FUNCTION_BLOCK fb_operationElecylinder
VAR_INPUT
END_VAR
VAR_OUTPUT
END_VAR
VAR
	SFCInit: bool;
	TranPosDone: BOOL;
	TranNegDone: BOOL;
	SamplePosDone: BOOL;
	SampleNegDone: BOOL;
	TrayChangePosDone: BOOL;
	TrayChangeNegDone: BOOL;
	flgInitDone: BOOL;
	trn_RotaryNegDone: BOOL;
	trn_RotaryPosDone: BOOL;
	trn_flgInitDone: BOOL;
	var_process: INT;
END_VAR

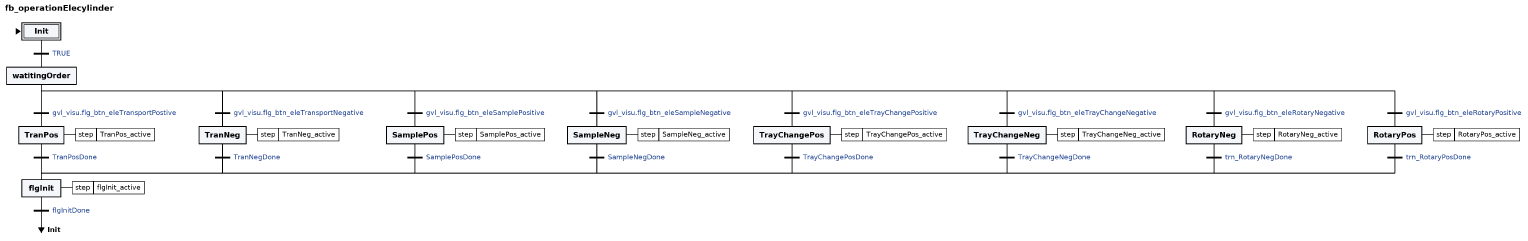
INITIAL_STEP Init:
END_STEP
TRANSITION FROM Init TO watitingOrder
    := TRUE;
END_TRANSITION
STEP watitingOrder:
END_STEP
TRANSITION FROM watitingOrder TO TranPos
    := gvl_visu.flg_btn_eleTransportPostive;
END_TRANSITION
STEP TranPos:
    TranPos_active(N);  // step action
END_STEP
TRANSITION FROM TranPos TO flgInit
    := TranPosDone;
END_TRANSITION
TRANSITION FROM watitingOrder TO TranNeg
    := gvl_visu.flg_btn_eleTransportNegative;
END_TRANSITION
STEP TranNeg:
    TranNeg_active(N);  // step action
END_STEP
TRANSITION FROM TranNeg TO flgInit
    := TranNegDone;
END_TRANSITION
TRANSITION FROM watitingOrder TO SamplePos
    := gvl_visu.flg_btn_eleSamplePositive;
END_TRANSITION
STEP SamplePos:
    SamplePos_active(N);  // step action
END_STEP
TRANSITION FROM SamplePos TO flgInit
    := SamplePosDone;
END_TRANSITION
TRANSITION FROM watitingOrder TO SampleNeg
    := gvl_visu.flg_btn_eleSampleNegative;
END_TRANSITION
STEP SampleNeg:
    SampleNeg_active(N);  // step action
END_STEP
TRANSITION FROM SampleNeg TO flgInit
    := SampleNegDone;
END_TRANSITION
TRANSITION FROM watitingOrder TO TrayChangePos
    := gvl_visu.flg_btn_eleTrayChangePositive;
END_TRANSITION
STEP TrayChangePos:
    TrayChangePos_active(N);  // step action
END_STEP
TRANSITION FROM TrayChangePos TO flgInit
    := TrayChangePosDone;
END_TRANSITION
TRANSITION FROM watitingOrder TO TrayChangeNeg
    := gvl_visu.flg_btn_eleTrayChangeNegative;
END_TRANSITION
STEP TrayChangeNeg:
    TrayChangeNeg_active(N);  // step action
END_STEP
TRANSITION FROM TrayChangeNeg TO flgInit
    := TrayChangeNegDone;
END_TRANSITION
TRANSITION FROM watitingOrder TO RotaryNeg
    := gvl_visu.flg_btn_eleRotaryNegative;
END_TRANSITION
STEP RotaryNeg:
    RotaryNeg_active(N);  // step action
END_STEP
TRANSITION FROM RotaryNeg TO flgInit
    := trn_RotaryNegDone;
END_TRANSITION
TRANSITION FROM watitingOrder TO RotaryPos
    := gvl_visu.flg_btn_eleRotaryPositive;
END_TRANSITION
STEP RotaryPos:
    RotaryPos_active(N);  // step action
END_STEP
TRANSITION FROM RotaryPos TO flgInit
    := trn_RotaryPosDone;
END_TRANSITION
STEP flgInit:
    flgInit_active(N);  // step action
END_STEP
TRANSITION FROM flgInit TO Init
    := flgInitDone;
END_TRANSITION

ACTION flgInit_active:
IF flgInit._x AND flgInit.x = FALSE THEN
	flgInitDone:= FALSE;
	gvl_visu.flg_btn_eleTransportPostive := FALSE;
	gvl_visu.flg_btn_eleTransportNegative := FALSE;
	gvl_visu.flg_btn_eleSamplePositive := FALSE;
	gvl_visu.flg_btn_eleSampleNegative := FALSE;
	gvl_visu.flg_btn_eleTrayChangePositive := FALSE;
	gvl_visu.flg_btn_eleTrayChangeNegative := FALSE;
	gvl_visu.flg_btn_eleRotaryPositive := FALSE;
	gvl_visu.flg_btn_eleRotaryNegative := FALSE;
ELSIF flgInit._x AND flgInit.x THEN
	flgInitDone := TRUE;
END_IF
END_ACTION

PROPERTY p_Init : bool
GET
p_init := THIS^.SFCInit;
END_GET
SET
THIS^.SFCInit := p_init;
END_SET
END_PROPERTY

ACTION RotaryNeg_active:
IF RotaryNeg._x AND RotaryNeg.x = FALSE THEN
	trn_RotaryNegDone := FALSE;
	gvl_elecylinder.fbi_axisRotary.in_flg_run := FALSE;
	gvl_elecylinder.fbi_axisRotary.in_var_moveMode := eP_eleMoveMode.eleA;
	var_process := 0;
ELSIF RotaryNeg._x AND RotaryNeg.x THEN
	CASE var_process OF
		0:
			gvl_elecylinder.fbi_axisRotary.in_flg_run := TRUE;
			var_process := 1;
		1:
			IF gvl_elecylinder.fbi_axisRotary.out_flg_Done THEN
				gvl_elecylinder.fbi_axisRotary.in_flg_run := FALSE;
				trn_RotaryNegDone := TRUE;
			END_IF
	END_CASE
END_IF
END_ACTION

ACTION RotaryPos_active:
IF RotaryPos._x AND RotaryPos.x = FALSE THEN
	trn_RotaryPosDone := FALSE;
	gvl_elecylinder.fbi_axisRotary.in_flg_run := FALSE;
	gvl_elecylinder.fbi_axisRotary.in_var_moveMode := eP_eleMoveMode.eleB;
	var_process := 0;
ELSIF RotaryPos._x AND RotaryPos.x THEN
	CASE var_process OF
		0:
			gvl_elecylinder.fbi_axisRotary.in_flg_run := TRUE;
			var_process :=1;
		1:
			IF gvl_elecylinder.fbi_axisRotary.out_flg_Done THEN
				gvl_elecylinder.fbi_axisRotary.in_flg_run := FALSE;
				trn_RotaryPosDone := TRUE;
			END_IF
	END_CASE
END_IF
END_ACTION

ACTION SampleNeg_active:
IF SampleNeg._x AND SampleNeg.x = FALSE THEN
	SampleNegDone := FALSE;
	gvl_elecylinder.fbi_axisSample.in_flg_run := FALSE;
	gvl_elecylinder.fbi_axisSample.in_var_moveMode := eP_eleMoveMode.eleA;
	var_process := 0;
ELSIF SampleNeg._x AND SampleNeg.x THEN
	CASE var_process OF
		0:
			gvl_elecylinder.fbi_axisSample.in_flg_run := TRUE;
			var_process := 1;
		1:
			IF gvl_elecylinder.fbi_axisSample.out_flg_Done THEN
				gvl_elecylinder.fbi_axisSample.in_flg_run := FALSE;
				SampleNegDone := TRUE;
			END_IF
	END_CASE
END_IF
END_ACTION

ACTION SamplePos_active:
IF SamplePos._x AND SamplePos.x = FALSE THEN
	SamplePosDone := FALSE;
	gvl_elecylinder.fbi_axisSample.in_flg_run := FALSE;
	gvl_elecylinder.fbi_axisSample.in_var_moveMode := eP_eleMoveMode.eleB;
	var_process := 0;
ELSIF SamplePos._x AND SamplePos.x THEN
	CASE var_process OF
		0:
			gvl_elecylinder.fbi_axisSample.in_flg_run := TRUE;
			var_process := 1;
		1:
			IF gvl_elecylinder.fbi_axisSample.out_flg_Done THEN
				gvl_elecylinder.fbi_axisSample.in_flg_run := FALSE;
				SamplePosDone := TRUE;
			END_IF
	END_CASE
END_IF
END_ACTION

ACTION TranNeg_active:
IF TranNeg._x AND TranNeg.x = FALSE THEN
	TranNegDone := FALSE;
	gvl_elecylinder.fbi_axisTransport.in_flg_run := FALSE;
	gvl_elecylinder.fbi_axisTransport.in_var_moveMode := eP_eleMoveMode.eleA;
	var_process := 0;
ELSIF TranNeg._x AND TranNeg.x THEN
	CASE var_process OF
		0:
			gvl_elecylinder.fbi_axisTransport.in_flg_run := TRUE;
			var_process := 1;
		1:
			IF gvl_elecylinder.fbi_axisTransport.out_flg_Done THEN
				gvl_elecylinder.fbi_axisTransport.in_flg_run := FALSE;
				TranNegDone := TRUE;
			END_IF
	END_CASE
END_IF
END_ACTION

ACTION TranPos_active:
IF TranPos._x AND TranPos.x = FALSE THEN
	TranPosDone := FALSE;
	gvl_elecylinder.fbi_axisTransport.in_flg_run := FALSE;
	gvl_elecylinder.fbi_axisTransport.in_var_moveMode := eP_eleMoveMode.eleB;
	var_process := 0;
ELSIF TranPos._x AND TranPos.x THEN
	CASE var_process OF
		0:
			gvl_elecylinder.fbi_axisTransport.in_flg_run := TRUE;
			var_process := 1;
		1:
			IF gvl_elecylinder.fbi_axisTransport.out_flg_Done THEN
				TranPosDone := TRUE;
			END_IF
	END_CASE
END_IF
END_ACTION

ACTION TrayChangeNeg_active:
IF TrayChangeNeg._x AND TrayChangeNeg.x = FALSE THEN
	TrayChangeNegDone := FALSE;
	gvl_elecylinder.fbi_axisTrayChange.in_flg_run := FALSE;
	gvl_elecylinder.fbi_axisTrayChange.in_var_moveMode := eP_eleMoveMode.eleA;
	var_process := 0;
ELSIF TrayChangeNeg._x AND TrayChangeNeg.x THEN
	CASE var_process OF
		0:
			gvl_axis.ref_z.Position := 50;
			gvl_axis.ref_z.Execute := TRUE;
			var_process := 1;
		1:
			IF gvl_axis.ref_z.Done THEN
				gvl_axis.ref_z.Execute := FALSE;
				var_process := 2;
			END_IF
		2:
			gvl_elecylinder.fbi_axisTrayChange.in_flg_run := TRUE;
			var_process := 3;
		3:
			IF gvl_elecylinder.fbi_axisTrayChange.out_flg_Done THEN
				gvl_elecylinder.fbi_axisTrayChange.in_flg_run := FALSE;
				TrayChangeNegDone := TRUE;
			END_IF
	END_CASE
END_IF
END_ACTION

ACTION TrayChangePos_active:
IF TrayChangePos._x AND TrayChangePos.x = FALSE THEN
	TrayChangePosDone := FALSE;
	gvl_elecylinder.fbi_axisTrayChange.in_flg_run := FALSE;
	gvl_elecylinder.fbi_axisTrayChange.in_var_moveMode := eP_eleMoveMode.eleB;
	var_process := 0;
ELSIF TrayChangePos._x AND TrayChangePos.x THEN
	CASE var_process OF
		0:
			gvl_axis.ref_z.Position := 50;
			gvl_axis.ref_z.Execute := TRUE;
			var_process := 1;
		1:
			IF gvl_axis.ref_z.Done THEN
				gvl_axis.ref_z.Execute := FALSE;
				var_process := 2;
			END_IF
		2:
			gvl_elecylinder.fbi_axisTrayChange.in_flg_run := TRUE;
			var_process := 3;
		3:
			IF gvl_elecylinder.fbi_axisTrayChange.out_flg_Done THEN
				gvl_elecylinder.fbi_axisTrayChange.in_flg_run := FALSE;
				TrayChangePosDone := TRUE;
			END_IF
	END_CASE
END_IF
END_ACTION

END_FUNCTION_BLOCK

(* stored: Version 1.1.0.1, ProductVersion 3.1.4024.11
   POU fb_operationElecylinder: Id {8ab1ae77-5bd3-40f0-99eb-fbf8e8064b36}, SpecialFunc None
   Action flgInit_active: Id {0b557403-70c8-4a74-b152-b2d0f9a2bd11}
   Property p_Init: Id {3c903e3c-02f6-4d30-86f8-53522214ca69}
   Get Get: Id {284f7822-1ff8-4e71-912d-44dc15521b76}
   Set Set: Id {0c610a4f-9c74-4baa-94d2-f11d079ccb92}
   Action RotaryNeg_active: Id {655d7f87-64fe-4f4c-8549-6d9b63c44ad6}
   Action RotaryPos_active: Id {b6866a1a-5afa-4ea8-84ac-c263eb9f8780}
   Action SampleNeg_active: Id {8169fc59-5f75-49ef-86f4-a06d8821b879}
   Action SamplePos_active: Id {b12f5653-50e1-46c5-9a47-baed4eb07751}
   Action TranNeg_active: Id {773d5a33-5f5c-45d0-9843-d859ad107dd9}
   Action TranPos_active: Id {1eb139fd-1d82-4c75-9ec7-ccbbfd23e3e0}
   Action TrayChangeNeg_active: Id {fadf5834-3bcc-4eb8-afc0-d09e629c6011}
   Action TrayChangePos_active: Id {26960138-7100-4c67-b13e-b71b03cefd06} *)
